# EPICS substitutions: ThingyApp/Db/aggregator.substitutions
file "bridge.template" {

# NodeID for the bridge Thingy = MAX_NODES

pattern { Sys,	Dev	}

{ "XF:10IDB",	"{THINGY:AGGREGATOR}"}

}
